FUNCTION_BLOCK Desidratacao (* Composite Function Block Type *)
  (* Standard: 61499-2 *)
  (* Version 0.5, 11/05/2026, Desidratacao de Lodo (Sec 4.8 EF). Refs: P&ID HID-PE-DE-ETE-FLX-002 R1 02/10/25; MD-35525-VCE-001 Rev.0 (2x SKID VSD-1200, Modbus PV-35525 IP 192.168.0.10 W:4001/4002 R:4005-4016); MD-36142-VCE-001 Rev.A (1x SKID VIB-3000 + 2 dosadoras M4/M5 internas, Modbus PV-36142 IP 192.168.0.10 W:4001/4002 R:4005-4019); Anexo I BIA-PC-RP-ETE-REL-007 sec 2.5.5-2.5.9. v0.3: top-level CAT (plcStart + IThis + SYMLINKMULTIVARDST). v0.4: SV_900_01/02/03 tipo corrigido para Valvula_Saida_Digital (sao solenoides); CPress3, VA_900_13, FT_900_06 marcados FUTURO. v0.5: SV_900_01..09 sao do Booster Lavagem 900-BR-01/02 (linha A.C.G. Agua Cinza Geral, Ø3/4 pol) - operacao MANUAL via faceplate individual de cada valvula no supervisorio (sem automacao). SV_900_01/02/03 = limpeza antes das BO_900_01/02/03 (sucção das bombas helicoidais). SV_900_04/05 = limpeza C-Press 1 (900-AD-01, 2 pontos). SV_900_06/07 = limpeza C-Press 2 (900-AD-02, 2 pontos). SV_900_08/09 = limpeza C-Press 3 (900-AD-03 FUTURO, 2 pontos). Adicionado conexoes IThis.E_RESET_FALHAS_PROCESSO -> SV_900_01..09.E_RESET_FALHA_PROCESSO para que o reset global tambem limpe falhas dessas valvulas. stsAutomatico default FALSE => modo manual permanente; cmdOnAutomatico/cmdOffAutomatico nao conectados. ARQUITETURA RESET: reset global IThis.cmdResetFalhas vai para BO_900_01/02/03 + BR_900_01/02 direto. Reset dos CPress vai por pinos individuais cmdResetFalha_CP1/2/3 (via Modbus PV-35525:4002). Preparador reset eh via faceplate propria (Preparador_Polimero_HMI tem cmdResetFalha interno). O supervisorio implementa 'Reset Geral' pulsando ambos os caminhos simultaneamente. BUGS DOCUMENTADOS EF (corrigir doc, nao codigo): Tabela 5 tem swap VA-12/VA-13 para AD-02/AD-03; basicCPressControl Sec 10 esta FISICAMENTE CORRETO conforme P&ID. Tabela 5 nao inclui VA-03/04/05 (descarga BO); basicCPressControl Sec 10/11 driva corretamente. TODOs: (1) cpRequest_1/2/3 e cpStop_1/2/3 do cPressControl pendentes (formula sugerida: cpRequest_X = CPress_X.stsFuncionamentoM1=1 AND CPress_X.stsEmergencia=0; cpStop_X = CPress_X.stsEmergencia<>0 OR CPress_X.stsAlarmeAcionado_critico). (2) Interlock LIT_900_01/02 (tanques estocagem) para bloqueio BO em baixo nivel (usar SYMLINKMULTIVARDST do CAT Estocagem_Lodo). *)
  PACKAGE Hidryco.HidrycoLib;
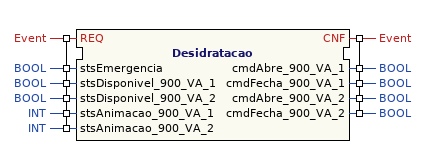
  EVENT_INPUT
    REQ WITH stsDisponivel_900_VA_1, stsDisponivel_900_VA_2, stsAnimacao_900_VA_1, stsAnimacao_900_VA_2, stsEmergencia;
  END_EVENT
  EVENT_OUTPUT
    CNF WITH cmdAbre_900_VA_1, cmdFecha_900_VA_1, cmdAbre_900_VA_2, cmdFecha_900_VA_2;
  END_EVENT
  VAR_INPUT
    stsEmergencia : BOOL;
    stsDisponivel_900_VA_1 : BOOL;
    stsDisponivel_900_VA_2 : BOOL;
    stsAnimacao_900_VA_1 : INT;
    stsAnimacao_900_VA_2 : INT;
  END_VAR
  VAR_OUTPUT
    cmdAbre_900_VA_1 : BOOL;
    cmdFecha_900_VA_1 : BOOL;
    cmdAbre_900_VA_2 : BOOL;
    cmdFecha_900_VA_2 : BOOL;
  END_VAR
  FBS
    BO_900_03 : Motor_Inversor_Automatico_Unico; (* Bomba Helicoidal alimentacao C-Press (3.7 kW). Revezamento 2+1. *)
    BO_900_02 : Motor_Inversor_Automatico_Unico; (* Bomba Helicoidal alimentacao C-Press (3.7 kW). Revezamento 2+1. *)
    BO_900_01 : Motor_Inversor_Automatico_Unico; (* Bomba Helicoidal alimentacao C-Press (3.7 kW, 35.25 m3/h). Revezamento 2+1. *)
    CPress1 : CPress; (* SKID Vibropac VSD-1200 (900-AD-01, PV-35525). Modbus TCP/IP. Status via SYMLINK interno. *)
    CPress2 : CPress; (* SKID Vibropac VSD-1200 (900-AD-02, PV-35525). Modbus TCP/IP. *)
    CPress3 : CPress; (* FUTURO (900-AD-03) conforme P&ID R1 02/10/25 *)
    Preparador_Polimero1 : Preparador_Polimero; (* SKID VIB-3000 (PV-36142). Integra via Modbus TCP/IP 192.168.0.10. Reset/Emergencia via faceplate propria. *)
    BR_900_01 : Motor_Inversor_Automatico_Unico; (* Booster Lavagem (7.35 kW, 2.5 m3/h @ 35 mca). MANUAL-ONLY conforme EF 4.8.3. *)
    BR_900_02 : Motor_Inversor_Automatico_Unico; (* Booster Lavagem (7.35 kW). Reserva. MANUAL-ONLY conforme EF 4.8.3. *)
    SV_900_03 : Valvula_Saida_Digital; (* Solenoide Booster Lavagem - antes da bomba BO_900_03 (manual via faceplate) *)
    SV_900_02 : Valvula_Saida_Digital; (* Solenoide Booster Lavagem - antes da bomba BO_900_02 (manual via faceplate) *)
    SV_900_01 : Valvula_Saida_Digital; (* Solenoide Booster Lavagem - antes da bomba BO_900_01 (manual via faceplate) *)
    VA_900_03 : Equipamento_On_Off;
    VA_900_04 : Equipamento_On_Off;
    VA_900_05 : Equipamento_On_Off;
    VA_900_08 : Equipamento_On_Off;
    VA_900_13 : Equipamento_On_Off; (* FUTURO (alimentacao 900-AD-03) conforme P&ID R1 02/10/25 *)
    VA_900_07 : Equipamento_On_Off;
    VA_900_12 : Equipamento_On_Off;
    VA_900_06 : Equipamento_On_Off;
    VA_900_11 : Equipamento_On_Off;
    VA_900_10 : Equipamento_On_Off;
    VA_900_09 : Equipamento_On_Off;
    FT_900_03 : Sensor_Comunicacao;
    FT_900_02 : Sensor_Comunicacao;
    FT_900_01 : Sensor_Comunicacao;
    SV_900_04 : Valvula_Saida_Digital; (* Solenoide Booster Lavagem - C-Press 1 (manual, ponto 1) *)
    SV_900_06 : Valvula_Saida_Digital; (* Solenoide Booster Lavagem - C-Press 2 (manual, ponto 1) *)
    SV_900_08 : Valvula_Saida_Digital; (* Solenoide Booster Lavagem - C-Press 3 (manual, ponto 1) - FUTURO *)
    plcStart1 : plcStart(Prio := 5);
    IThis : Desidratacao_HMI(QI := TRUE);
    SYMLINKMULTIVARDST1 : SYMLINKMULTIVARDST_1559B0FF8170C9BA0(QI := TRUE, NAME1 := '$${PATH}stsEmergencia'); {SET_ATTRIBUTE(Configuration.GenericFBType.InterfaceParams, Runtime.System#I:=1;VALUE${I$}:BOOL)}
    FT_900_07 : Sensor_Comunicacao;
    FT_QT_01 : Sensor_Comunicacao;
  END_FBS
  EVENT_CONNECTIONS
    plcStart1.FIRST_INIT TO IThis.A0000001000000A1;
    plcStart1.REDO_INIT TO IThis.A0000001000000A1;
    IThis.A0000001000000B1 TO SYMLINKMULTIVARDST1.INIT;
    SYMLINKMULTIVARDST1.INITO TO plcStart1.ACK_FIRST;
    IThis.A0000001000000B1 TO CPress1.INIT;
    IThis.A0000001000000B1 TO CPress2.INIT;
    IThis.A0000001000000B1 TO CPress3.INIT;
    IThis.A0000001000000B1 TO Preparador_Polimero1.INIT;
    IThis.A0000001000000B2 TO BO_900_01.E_RESET_FALHA_PROCESSO;
    IThis.A0000001000000B2 TO BO_900_02.E_RESET_FALHA_PROCESSO;
    IThis.A0000001000000B2 TO BO_900_03.E_RESET_FALHA_PROCESSO;
    IThis.A0000001000000B2 TO BR_900_01.E_RESET_FALHA_PROCESSO;
    IThis.A0000001000000B2 TO BR_900_02.E_RESET_FALHA_PROCESSO;
    IThis.A0000001000000B3 TO CPress1.REQ;
    IThis.A0000001000000B3 TO CPress2.REQ;
    IThis.A0000001000000B3 TO CPress3.REQ;
    IThis.A0000001000000B3 TO Preparador_Polimero1.REQ;
    IThis.A0000001000000B2 TO SV_900_01.E_RESET_FALHA_PROCESSO;
    IThis.A0000001000000B2 TO SV_900_02.E_RESET_FALHA_PROCESSO;
    IThis.A0000001000000B2 TO SV_900_03.E_RESET_FALHA_PROCESSO;
    IThis.A0000001000000B2 TO SV_900_04.E_RESET_FALHA_PROCESSO;
    IThis.A0000001000000B2 TO SV_900_06.E_RESET_FALHA_PROCESSO;
    IThis.A0000001000000B2 TO SV_900_08.E_RESET_FALHA_PROCESSO;
    REQ TO VA_900_04.REQ;
    REQ TO VA_900_05.REQ;
    REQ TO VA_900_03.REQ;
    REQ TO BO_900_03.REQ;
    REQ TO BO_900_02.REQ;
    REQ TO BO_900_01.REQ;
    REQ TO VA_900_06.REQ;
    REQ TO VA_900_07.REQ;
    REQ TO VA_900_08.REQ;
    REQ TO VA_900_13.REQ;
    REQ TO VA_900_11.REQ;
    REQ TO VA_900_09.REQ;
    REQ TO VA_900_10.REQ;
    REQ TO VA_900_12.REQ;
  END_CONNECTIONS
  DATA_CONNECTIONS
    IThis.A0000001000000D3 TO BO_900_01.cmdResetFalhas;
    IThis.A0000001000000D3 TO BO_900_02.cmdResetFalhas;
    IThis.A0000001000000D3 TO BO_900_03.cmdResetFalhas;
    IThis.A0000001000000D3 TO BR_900_01.cmdResetFalhas;
    IThis.A0000001000000D3 TO BR_900_02.cmdResetFalhas;
    IThis.A0000001000000D9 TO CPress1.cmdLigaDesligaCicloRemoto;
    IThis.A0000001000000DA TO CPress2.cmdLigaDesligaCicloRemoto;
    IThis.A0000001000000DB TO CPress3.cmdLigaDesligaCicloRemoto;
    IThis.A0000001000000DC TO CPress1.cmdResetFalha;
    IThis.A0000001000000DD TO CPress2.cmdResetFalha;
    IThis.A0000001000000DE TO CPress3.cmdResetFalha;
    IThis.A0000001000000DF TO Preparador_Polimero1.acmAutomatico;
    IThis.A0000001000000E0 TO Preparador_Polimero1.stsAutomatico;
    stsEmergencia TO VA_900_03.E74E49E48343E6DC;
    stsEmergencia TO VA_900_04.E74E49E48343E6DC;
    stsEmergencia TO VA_900_05.E74E49E48343E6DC;
    stsEmergencia TO VA_900_08.E74E49E48343E6DC;
    stsEmergencia TO VA_900_07.E74E49E48343E6DC;
    stsEmergencia TO VA_900_06.E74E49E48343E6DC;
    stsEmergencia TO VA_900_11.E74E49E48343E6DC;
    stsEmergencia TO VA_900_09.E74E49E48343E6DC;
    stsEmergencia TO VA_900_10.E74E49E48343E6DC;
    stsEmergencia TO VA_900_13.E74E49E48343E6DC;
    stsEmergencia TO VA_900_12.E74E49E48343E6DC;
    stsEmergencia TO BO_900_01.stsEmergencia;
    stsEmergencia TO BO_900_02.stsEmergencia;
    stsEmergencia TO BO_900_03.stsEmergencia;
  END_CONNECTIONS
END_FUNCTION_BLOCK
